// TIA Portal V20 export
DATA_BLOCK "instGetMotorstarterSignals"   // DB91
// stored: InstanceOfName GetMotorstarterSignals, InstanceOfType FB
"GetMotorstarterSignals"
   // VAR_INPUT
   //    Et200SpMotorstarterInterfaceAllUnits { ExternalAccessible := 'False'; ExternalVisible := 'False'; ExternalWritable := 'False'} : Array[0.."NO_OF_UNITS"] of "typeEmMotorStarterInterface";
   //    numberOfMS : USInt := 1;
   // END_VAR
   // VAR_OUTPUT
   //    selectedUnit : USInt := 1;
   //    selectedEM : USInt := 6;
   //    error : Word := 16#7001;
   // END_VAR
   // VAR_IN_OUT
   //    Et200SpMotorstarterInterfaceHmi : "typeEt200SpMotorstarterInterfaceHmi";
   // END_VAR
   // VAR
   //    statSelectedEMMotorStarter : USInt := 6;
   //    statSelectedUnitMotorStarter : USInt := 1;
   // END_VAR
BEGIN
   Et200SpMotorstarterInterfaceAllUnits[0].EMmotorstarter[0].et200SpMotorstarterCurrent[0..1] := 0.0;
   Et200SpMotorstarterInterfaceAllUnits[0].EMmotorstarter[1].et200SpMotorstarterCurrent[0..1] := 0.0;
   Et200SpMotorstarterInterfaceAllUnits[0].EMmotorstarter[2].et200SpMotorstarterCurrent[0..1] := 0.0;
   Et200SpMotorstarterInterfaceAllUnits[0].EMmotorstarter[3].et200SpMotorstarterCurrent[0..1] := 0.0;
   Et200SpMotorstarterInterfaceAllUnits[0].EMmotorstarter[4].et200SpMotorstarterCurrent[0..1] := 0.0;
   Et200SpMotorstarterInterfaceAllUnits[0].EMmotorstarter[5].et200SpMotorstarterCurrent[0..1] := 0.0;
   Et200SpMotorstarterInterfaceAllUnits[0].EMmotorstarter[6].et200SpMotorstarterCurrent[0..1] := 0.0;
   Et200SpMotorstarterInterfaceAllUnits[0].EMmotorstarter[7].et200SpMotorstarterCurrent[0..1] := 0.0;
   Et200SpMotorstarterInterfaceAllUnits[0].EMmotorstarter[0].et200SpMotorstarterInputs[0..1].readyAutomatic := FALSE;
   Et200SpMotorstarterInterfaceAllUnits[0].EMmotorstarter[1].et200SpMotorstarterInputs[0..1].readyAutomatic := FALSE;
   Et200SpMotorstarterInterfaceAllUnits[0].EMmotorstarter[2].et200SpMotorstarterInputs[0..1].readyAutomatic := FALSE;
   Et200SpMotorstarterInterfaceAllUnits[0].EMmotorstarter[3].et200SpMotorstarterInputs[0..1].readyAutomatic := FALSE;
   Et200SpMotorstarterInterfaceAllUnits[0].EMmotorstarter[4].et200SpMotorstarterInputs[0..1].readyAutomatic := FALSE;
   Et200SpMotorstarterInterfaceAllUnits[0].EMmotorstarter[5].et200SpMotorstarterInputs[0..1].readyAutomatic := FALSE;
   Et200SpMotorstarterInterfaceAllUnits[0].EMmotorstarter[6].et200SpMotorstarterInputs[0..1].readyAutomatic := FALSE;
   Et200SpMotorstarterInterfaceAllUnits[0].EMmotorstarter[7].et200SpMotorstarterInputs[0..1].readyAutomatic := FALSE;
   Et200SpMotorstarterInterfaceAllUnits[0].EMmotorstarter[0].et200SpMotorstarterInputs[0..1].motorOn := FALSE;
   Et200SpMotorstarterInterfaceAllUnits[0].EMmotorstarter[1].et200SpMotorstarterInputs[0..1].motorOn := FALSE;
   Et200SpMotorstarterInterfaceAllUnits[0].EMmotorstarter[2].et200SpMotorstarterInputs[0..1].motorOn := FALSE;
   Et200SpMotorstarterInterfaceAllUnits[0].EMmotorstarter[3].et200SpMotorstarterInputs[0..1].motorOn := FALSE;
   Et200SpMotorstarterInterfaceAllUnits[0].EMmotorstarter[4].et200SpMotorstarterInputs[0..1].motorOn := FALSE;
   Et200SpMotorstarterInterfaceAllUnits[0].EMmotorstarter[5].et200SpMotorstarterInputs[0..1].motorOn := FALSE;
   Et200SpMotorstarterInterfaceAllUnits[0].EMmotorstarter[6].et200SpMotorstarterInputs[0..1].motorOn := FALSE;
   Et200SpMotorstarterInterfaceAllUnits[0].EMmotorstarter[7].et200SpMotorstarterInputs[0..1].motorOn := FALSE;
   Et200SpMotorstarterInterfaceAllUnits[0].EMmotorstarter[0].et200SpMotorstarterInputs[0..1].groupFault := FALSE;
   Et200SpMotorstarterInterfaceAllUnits[0].EMmotorstarter[1].et200SpMotorstarterInputs[0..1].groupFault := FALSE;
   Et200SpMotorstarterInterfaceAllUnits[0].EMmotorstarter[2].et200SpMotorstarterInputs[0..1].groupFault := FALSE;
   Et200SpMotorstarterInterfaceAllUnits[0].EMmotorstarter[3].et200SpMotorstarterInputs[0..1].groupFault := FALSE;
   Et200SpMotorstarterInterfaceAllUnits[0].EMmotorstarter[4].et200SpMotorstarterInputs[0..1].groupFault := FALSE;
   Et200SpMotorstarterInterfaceAllUnits[0].EMmotorstarter[5].et200SpMotorstarterInputs[0..1].groupFault := FALSE;
   Et200SpMotorstarterInterfaceAllUnits[0].EMmotorstarter[6].et200SpMotorstarterInputs[0..1].groupFault := FALSE;
   Et200SpMotorstarterInterfaceAllUnits[0].EMmotorstarter[7].et200SpMotorstarterInputs[0..1].groupFault := FALSE;
   Et200SpMotorstarterInterfaceAllUnits[0].EMmotorstarter[0].et200SpMotorstarterInputs[0..1].groupWarning := FALSE;
   Et200SpMotorstarterInterfaceAllUnits[0].EMmotorstarter[1].et200SpMotorstarterInputs[0..1].groupWarning := FALSE;
   Et200SpMotorstarterInterfaceAllUnits[0].EMmotorstarter[2].et200SpMotorstarterInputs[0..1].groupWarning := FALSE;
   Et200SpMotorstarterInterfaceAllUnits[0].EMmotorstarter[3].et200SpMotorstarterInputs[0..1].groupWarning := FALSE;
   Et200SpMotorstarterInterfaceAllUnits[0].EMmotorstarter[4].et200SpMotorstarterInputs[0..1].groupWarning := FALSE;
   Et200SpMotorstarterInterfaceAllUnits[0].EMmotorstarter[5].et200SpMotorstarterInputs[0..1].groupWarning := FALSE;
   Et200SpMotorstarterInterfaceAllUnits[0].EMmotorstarter[6].et200SpMotorstarterInputs[0..1].groupWarning := FALSE;
   Et200SpMotorstarterInterfaceAllUnits[0].EMmotorstarter[7].et200SpMotorstarterInputs[0..1].groupWarning := FALSE;
   Et200SpMotorstarterInterfaceAllUnits[0].EMmotorstarter[0].et200SpMotorstarterInputs[0..1].input1 := FALSE;
   Et200SpMotorstarterInterfaceAllUnits[0].EMmotorstarter[1].et200SpMotorstarterInputs[0..1].input1 := FALSE;
   Et200SpMotorstarterInterfaceAllUnits[0].EMmotorstarter[2].et200SpMotorstarterInputs[0..1].input1 := FALSE;
   Et200SpMotorstarterInterfaceAllUnits[0].EMmotorstarter[3].et200SpMotorstarterInputs[0..1].input1 := FALSE;
   Et200SpMotorstarterInterfaceAllUnits[0].EMmotorstarter[4].et200SpMotorstarterInputs[0..1].input1 := FALSE;
   Et200SpMotorstarterInterfaceAllUnits[0].EMmotorstarter[5].et200SpMotorstarterInputs[0..1].input1 := FALSE;
   Et200SpMotorstarterInterfaceAllUnits[0].EMmotorstarter[6].et200SpMotorstarterInputs[0..1].input1 := FALSE;
   Et200SpMotorstarterInterfaceAllUnits[0].EMmotorstarter[7].et200SpMotorstarterInputs[0..1].input1 := FALSE;
   Et200SpMotorstarterInterfaceAllUnits[0].EMmotorstarter[0].et200SpMotorstarterInputs[0..1].input2 := FALSE;
   Et200SpMotorstarterInterfaceAllUnits[0].EMmotorstarter[1].et200SpMotorstarterInputs[0..1].input2 := FALSE;
   Et200SpMotorstarterInterfaceAllUnits[0].EMmotorstarter[2].et200SpMotorstarterInputs[0..1].input2 := FALSE;
   Et200SpMotorstarterInterfaceAllUnits[0].EMmotorstarter[3].et200SpMotorstarterInputs[0..1].input2 := FALSE;
   Et200SpMotorstarterInterfaceAllUnits[0].EMmotorstarter[4].et200SpMotorstarterInputs[0..1].input2 := FALSE;
   Et200SpMotorstarterInterfaceAllUnits[0].EMmotorstarter[5].et200SpMotorstarterInputs[0..1].input2 := FALSE;
   Et200SpMotorstarterInterfaceAllUnits[0].EMmotorstarter[6].et200SpMotorstarterInputs[0..1].input2 := FALSE;
   Et200SpMotorstarterInterfaceAllUnits[0].EMmotorstarter[7].et200SpMotorstarterInputs[0..1].input2 := FALSE;
   Et200SpMotorstarterInterfaceAllUnits[0].EMmotorstarter[0].et200SpMotorstarterInputs[0..1].input3 := FALSE;
   Et200SpMotorstarterInterfaceAllUnits[0].EMmotorstarter[1].et200SpMotorstarterInputs[0..1].input3 := FALSE;
   Et200SpMotorstarterInterfaceAllUnits[0].EMmotorstarter[2].et200SpMotorstarterInputs[0..1].input3 := FALSE;
   Et200SpMotorstarterInterfaceAllUnits[0].EMmotorstarter[3].et200SpMotorstarterInputs[0..1].input3 := FALSE;
   Et200SpMotorstarterInterfaceAllUnits[0].EMmotorstarter[4].et200SpMotorstarterInputs[0..1].input3 := FALSE;
   Et200SpMotorstarterInterfaceAllUnits[0].EMmotorstarter[5].et200SpMotorstarterInputs[0..1].input3 := FALSE;
   Et200SpMotorstarterInterfaceAllUnits[0].EMmotorstarter[6].et200SpMotorstarterInputs[0..1].input3 := FALSE;
   Et200SpMotorstarterInterfaceAllUnits[0].EMmotorstarter[7].et200SpMotorstarterInputs[0..1].input3 := FALSE;
   Et200SpMotorstarterInterfaceAllUnits[0].EMmotorstarter[0].et200SpMotorstarterInputs[0..1].inputLocalCtrl := FALSE;
   Et200SpMotorstarterInterfaceAllUnits[0].EMmotorstarter[1].et200SpMotorstarterInputs[0..1].inputLocalCtrl := FALSE;
   Et200SpMotorstarterInterfaceAllUnits[0].EMmotorstarter[2].et200SpMotorstarterInputs[0..1].inputLocalCtrl := FALSE;
   Et200SpMotorstarterInterfaceAllUnits[0].EMmotorstarter[3].et200SpMotorstarterInputs[0..1].inputLocalCtrl := FALSE;
   Et200SpMotorstarterInterfaceAllUnits[0].EMmotorstarter[4].et200SpMotorstarterInputs[0..1].inputLocalCtrl := FALSE;
   Et200SpMotorstarterInterfaceAllUnits[0].EMmotorstarter[5].et200SpMotorstarterInputs[0..1].inputLocalCtrl := FALSE;
   Et200SpMotorstarterInterfaceAllUnits[0].EMmotorstarter[6].et200SpMotorstarterInputs[0..1].inputLocalCtrl := FALSE;
   Et200SpMotorstarterInterfaceAllUnits[0].EMmotorstarter[7].et200SpMotorstarterInputs[0..1].inputLocalCtrl := FALSE;
   Et200SpMotorstarterInterfaceAllUnits[0].EMmotorstarter[0].et200SpMotorstarterInputs[0..1].iActBit0 := FALSE;
   Et200SpMotorstarterInterfaceAllUnits[0].EMmotorstarter[1].et200SpMotorstarterInputs[0..1].iActBit0 := FALSE;
   Et200SpMotorstarterInterfaceAllUnits[0].EMmotorstarter[2].et200SpMotorstarterInputs[0..1].iActBit0 := FALSE;
   Et200SpMotorstarterInterfaceAllUnits[0].EMmotorstarter[3].et200SpMotorstarterInputs[0..1].iActBit0 := FALSE;
   Et200SpMotorstarterInterfaceAllUnits[0].EMmotorstarter[4].et200SpMotorstarterInputs[0..1].iActBit0 := FALSE;
   Et200SpMotorstarterInterfaceAllUnits[0].EMmotorstarter[5].et200SpMotorstarterInputs[0..1].iActBit0 := FALSE;
   Et200SpMotorstarterInterfaceAllUnits[0].EMmotorstarter[6].et200SpMotorstarterInputs[0..1].iActBit0 := FALSE;
   Et200SpMotorstarterInterfaceAllUnits[0].EMmotorstarter[7].et200SpMotorstarterInputs[0..1].iActBit0 := FALSE;
   Et200SpMotorstarterInterfaceAllUnits[0].EMmotorstarter[0].et200SpMotorstarterInputs[0..1].iActBit1 := FALSE;
   Et200SpMotorstarterInterfaceAllUnits[0].EMmotorstarter[1].et200SpMotorstarterInputs[0..1].iActBit1 := FALSE;
   Et200SpMotorstarterInterfaceAllUnits[0].EMmotorstarter[2].et200SpMotorstarterInputs[0..1].iActBit1 := FALSE;
   Et200SpMotorstarterInterfaceAllUnits[0].EMmotorstarter[3].et200SpMotorstarterInputs[0..1].iActBit1 := FALSE;
   Et200SpMotorstarterInterfaceAllUnits[0].EMmotorstarter[4].et200SpMotorstarterInputs[0..1].iActBit1 := FALSE;
   Et200SpMotorstarterInterfaceAllUnits[0].EMmotorstarter[5].et200SpMotorstarterInputs[0..1].iActBit1 := FALSE;
   Et200SpMotorstarterInterfaceAllUnits[0].EMmotorstarter[6].et200SpMotorstarterInputs[0..1].iActBit1 := FALSE;
   Et200SpMotorstarterInterfaceAllUnits[0].EMmotorstarter[7].et200SpMotorstarterInputs[0..1].iActBit1 := FALSE;
   Et200SpMotorstarterInterfaceAllUnits[0].EMmotorstarter[0].et200SpMotorstarterInputs[0..1].iActBit2 := FALSE;
   Et200SpMotorstarterInterfaceAllUnits[0].EMmotorstarter[1].et200SpMotorstarterInputs[0..1].iActBit2 := FALSE;
   Et200SpMotorstarterInterfaceAllUnits[0].EMmotorstarter[2].et200SpMotorstarterInputs[0..1].iActBit2 := FALSE;
   Et200SpMotorstarterInterfaceAllUnits[0].EMmotorstarter[3].et200SpMotorstarterInputs[0..1].iActBit2 := FALSE;
   Et200SpMotorstarterInterfaceAllUnits[0].EMmotorstarter[4].et200SpMotorstarterInputs[0..1].iActBit2 := FALSE;
   Et200SpMotorstarterInterfaceAllUnits[0].EMmotorstarter[5].et200SpMotorstarterInputs[0..1].iActBit2 := FALSE;
   Et200SpMotorstarterInterfaceAllUnits[0].EMmotorstarter[6].et200SpMotorstarterInputs[0..1].iActBit2 := FALSE;
   Et200SpMotorstarterInterfaceAllUnits[0].EMmotorstarter[7].et200SpMotorstarterInputs[0..1].iActBit2 := FALSE;
   Et200SpMotorstarterInterfaceAllUnits[0].EMmotorstarter[0].et200SpMotorstarterInputs[0..1].iActBit3 := FALSE;
   Et200SpMotorstarterInterfaceAllUnits[0].EMmotorstarter[1].et200SpMotorstarterInputs[0..1].iActBit3 := FALSE;
   Et200SpMotorstarterInterfaceAllUnits[0].EMmotorstarter[2].et200SpMotorstarterInputs[0..1].iActBit3 := FALSE;
   Et200SpMotorstarterInterfaceAllUnits[0].EMmotorstarter[3].et200SpMotorstarterInputs[0..1].iActBit3 := FALSE;
   Et200SpMotorstarterInterfaceAllUnits[0].EMmotorstarter[4].et200SpMotorstarterInputs[0..1].iActBit3 := FALSE;
   Et200SpMotorstarterInterfaceAllUnits[0].EMmotorstarter[5].et200SpMotorstarterInputs[0..1].iActBit3 := FALSE;
   Et200SpMotorstarterInterfaceAllUnits[0].EMmotorstarter[6].et200SpMotorstarterInputs[0..1].iActBit3 := FALSE;
   Et200SpMotorstarterInterfaceAllUnits[0].EMmotorstarter[7].et200SpMotorstarterInputs[0..1].iActBit3 := FALSE;
   Et200SpMotorstarterInterfaceAllUnits[0].EMmotorstarter[0].et200SpMotorstarterInputs[0..1].iActBit4 := FALSE;
   Et200SpMotorstarterInterfaceAllUnits[0].EMmotorstarter[1].et200SpMotorstarterInputs[0..1].iActBit4 := FALSE;
   Et200SpMotorstarterInterfaceAllUnits[0].EMmotorstarter[2].et200SpMotorstarterInputs[0..1].iActBit4 := FALSE;
   Et200SpMotorstarterInterfaceAllUnits[0].EMmotorstarter[3].et200SpMotorstarterInputs[0..1].iActBit4 := FALSE;
   Et200SpMotorstarterInterfaceAllUnits[0].EMmotorstarter[4].et200SpMotorstarterInputs[0..1].iActBit4 := FALSE;
   Et200SpMotorstarterInterfaceAllUnits[0].EMmotorstarter[5].et200SpMotorstarterInputs[0..1].iActBit4 := FALSE;
   Et200SpMotorstarterInterfaceAllUnits[0].EMmotorstarter[6].et200SpMotorstarterInputs[0..1].iActBit4 := FALSE;
   Et200SpMotorstarterInterfaceAllUnits[0].EMmotorstarter[7].et200SpMotorstarterInputs[0..1].iActBit4 := FALSE;
   Et200SpMotorstarterInterfaceAllUnits[0].EMmotorstarter[0].et200SpMotorstarterInputs[0..1].iActBit5 := FALSE;
   Et200SpMotorstarterInterfaceAllUnits[0].EMmotorstarter[1].et200SpMotorstarterInputs[0..1].iActBit5 := FALSE;
   Et200SpMotorstarterInterfaceAllUnits[0].EMmotorstarter[2].et200SpMotorstarterInputs[0..1].iActBit5 := FALSE;
   Et200SpMotorstarterInterfaceAllUnits[0].EMmotorstarter[3].et200SpMotorstarterInputs[0..1].iActBit5 := FALSE;
   Et200SpMotorstarterInterfaceAllUnits[0].EMmotorstarter[4].et200SpMotorstarterInputs[0..1].iActBit5 := FALSE;
   Et200SpMotorstarterInterfaceAllUnits[0].EMmotorstarter[5].et200SpMotorstarterInputs[0..1].iActBit5 := FALSE;
   Et200SpMotorstarterInterfaceAllUnits[0].EMmotorstarter[6].et200SpMotorstarterInputs[0..1].iActBit5 := FALSE;
   Et200SpMotorstarterInterfaceAllUnits[0].EMmotorstarter[7].et200SpMotorstarterInputs[0..1].iActBit5 := FALSE;
   Et200SpMotorstarterInterfaceAllUnits[0].EMmotorstarter[0].et200SpMotorstarterInputs[0..1].manualOperating := FALSE;
   Et200SpMotorstarterInterfaceAllUnits[0].EMmotorstarter[1].et200SpMotorstarterInputs[0..1].manualOperating := FALSE;
   Et200SpMotorstarterInterfaceAllUnits[0].EMmotorstarter[2].et200SpMotorstarterInputs[0..1].manualOperating := FALSE;
   Et200SpMotorstarterInterfaceAllUnits[0].EMmotorstarter[3].et200SpMotorstarterInputs[0..1].manualOperating := FALSE;
   Et200SpMotorstarterInterfaceAllUnits[0].EMmotorstarter[4].et200SpMotorstarterInputs[0..1].manualOperating := FALSE;
   Et200SpMotorstarterInterfaceAllUnits[0].EMmotorstarter[5].et200SpMotorstarterInputs[0..1].manualOperating := FALSE;
   Et200SpMotorstarterInterfaceAllUnits[0].EMmotorstarter[6].et200SpMotorstarterInputs[0..1].manualOperating := FALSE;
   Et200SpMotorstarterInterfaceAllUnits[0].EMmotorstarter[7].et200SpMotorstarterInputs[0..1].manualOperating := FALSE;
   Et200SpMotorstarterInterfaceAllUnits[0].EMmotorstarter[0].et200SpMotorstarterInputs[0..1].spare1 := FALSE;
   Et200SpMotorstarterInterfaceAllUnits[0].EMmotorstarter[1].et200SpMotorstarterInputs[0..1].spare1 := FALSE;
   Et200SpMotorstarterInterfaceAllUnits[0].EMmotorstarter[2].et200SpMotorstarterInputs[0..1].spare1 := FALSE;
   Et200SpMotorstarterInterfaceAllUnits[0].EMmotorstarter[3].et200SpMotorstarterInputs[0..1].spare1 := FALSE;
   Et200SpMotorstarterInterfaceAllUnits[0].EMmotorstarter[4].et200SpMotorstarterInputs[0..1].spare1 := FALSE;
   Et200SpMotorstarterInterfaceAllUnits[0].EMmotorstarter[5].et200SpMotorstarterInputs[0..1].spare1 := FALSE;
   Et200SpMotorstarterInterfaceAllUnits[0].EMmotorstarter[6].et200SpMotorstarterInputs[0..1].spare1 := FALSE;
   Et200SpMotorstarterInterfaceAllUnits[0].EMmotorstarter[7].et200SpMotorstarterInputs[0..1].spare1 := FALSE;
   Et200SpMotorstarterInterfaceAllUnits[0].EMmotorstarter[0].et200SpMotorstarterInputs[0..1].readyStartOn := FALSE;
   Et200SpMotorstarterInterfaceAllUnits[0].EMmotorstarter[1].et200SpMotorstarterInputs[0..1].readyStartOn := FALSE;
   Et200SpMotorstarterInterfaceAllUnits[0].EMmotorstarter[2].et200SpMotorstarterInputs[0..1].readyStartOn := FALSE;
   Et200SpMotorstarterInterfaceAllUnits[0].EMmotorstarter[3].et200SpMotorstarterInputs[0..1].readyStartOn := FALSE;
   Et200SpMotorstarterInterfaceAllUnits[0].EMmotorstarter[4].et200SpMotorstarterInputs[0..1].readyStartOn := FALSE;
   Et200SpMotorstarterInterfaceAllUnits[0].EMmotorstarter[5].et200SpMotorstarterInputs[0..1].readyStartOn := FALSE;
   Et200SpMotorstarterInterfaceAllUnits[0].EMmotorstarter[6].et200SpMotorstarterInputs[0..1].readyStartOn := FALSE;
   Et200SpMotorstarterInterfaceAllUnits[0].EMmotorstarter[7].et200SpMotorstarterInputs[0..1].readyStartOn := FALSE;
   Et200SpMotorstarterInterfaceAllUnits[0].EMmotorstarter[0].et200SpMotorstarterInputs[0..1].motorOnRight := FALSE;
   Et200SpMotorstarterInterfaceAllUnits[0].EMmotorstarter[1].et200SpMotorstarterInputs[0..1].motorOnRight := FALSE;
   Et200SpMotorstarterInterfaceAllUnits[0].EMmotorstarter[2].et200SpMotorstarterInputs[0..1].motorOnRight := FALSE;
   Et200SpMotorstarterInterfaceAllUnits[0].EMmotorstarter[3].et200SpMotorstarterInputs[0..1].motorOnRight := FALSE;
   Et200SpMotorstarterInterfaceAllUnits[0].EMmotorstarter[4].et200SpMotorstarterInputs[0..1].motorOnRight := FALSE;
   Et200SpMotorstarterInterfaceAllUnits[0].EMmotorstarter[5].et200SpMotorstarterInputs[0..1].motorOnRight := FALSE;
   Et200SpMotorstarterInterfaceAllUnits[0].EMmotorstarter[6].et200SpMotorstarterInputs[0..1].motorOnRight := FALSE;
   Et200SpMotorstarterInterfaceAllUnits[0].EMmotorstarter[7].et200SpMotorstarterInputs[0..1].motorOnRight := FALSE;
   Et200SpMotorstarterInterfaceAllUnits[0].EMmotorstarter[0].et200SpMotorstarterInputs[0..1].motorOnLeft := FALSE;
   Et200SpMotorstarterInterfaceAllUnits[0].EMmotorstarter[1].et200SpMotorstarterInputs[0..1].motorOnLeft := FALSE;
   Et200SpMotorstarterInterfaceAllUnits[0].EMmotorstarter[2].et200SpMotorstarterInputs[0..1].motorOnLeft := FALSE;
   Et200SpMotorstarterInterfaceAllUnits[0].EMmotorstarter[3].et200SpMotorstarterInputs[0..1].motorOnLeft := FALSE;
   Et200SpMotorstarterInterfaceAllUnits[0].EMmotorstarter[4].et200SpMotorstarterInputs[0..1].motorOnLeft := FALSE;
   Et200SpMotorstarterInterfaceAllUnits[0].EMmotorstarter[5].et200SpMotorstarterInputs[0..1].motorOnLeft := FALSE;
   Et200SpMotorstarterInterfaceAllUnits[0].EMmotorstarter[6].et200SpMotorstarterInputs[0..1].motorOnLeft := FALSE;
   Et200SpMotorstarterInterfaceAllUnits[0].EMmotorstarter[7].et200SpMotorstarterInputs[0..1].motorOnLeft := FALSE;
   Et200SpMotorstarterInterfaceAllUnits[0].EMmotorstarter[0].et200SpMotorstarterInputs[0..1].quickstopActive := FALSE;
   Et200SpMotorstarterInterfaceAllUnits[0].EMmotorstarter[1].et200SpMotorstarterInputs[0..1].quickstopActive := FALSE;
   Et200SpMotorstarterInterfaceAllUnits[0].EMmotorstarter[2].et200SpMotorstarterInputs[0..1].quickstopActive := FALSE;
   Et200SpMotorstarterInterfaceAllUnits[0].EMmotorstarter[3].et200SpMotorstarterInputs[0..1].quickstopActive := FALSE;
   Et200SpMotorstarterInterfaceAllUnits[0].EMmotorstarter[4].et200SpMotorstarterInputs[0..1].quickstopActive := FALSE;
   Et200SpMotorstarterInterfaceAllUnits[0].EMmotorstarter[5].et200SpMotorstarterInputs[0..1].quickstopActive := FALSE;
   Et200SpMotorstarterInterfaceAllUnits[0].EMmotorstarter[6].et200SpMotorstarterInputs[0..1].quickstopActive := FALSE;
   Et200SpMotorstarterInterfaceAllUnits[0].EMmotorstarter[7].et200SpMotorstarterInputs[0..1].quickstopActive := FALSE;
   Et200SpMotorstarterInterfaceAllUnits[0].EMmotorstarter[0].et200SpMotorstarterInputs[0..1].energySaving := FALSE;
   Et200SpMotorstarterInterfaceAllUnits[0].EMmotorstarter[1].et200SpMotorstarterInputs[0..1].energySaving := FALSE;
   Et200SpMotorstarterInterfaceAllUnits[0].EMmotorstarter[2].et200SpMotorstarterInputs[0..1].energySaving := FALSE;
   Et200SpMotorstarterInterfaceAllUnits[0].EMmotorstarter[3].et200SpMotorstarterInputs[0..1].energySaving := FALSE;
   Et200SpMotorstarterInterfaceAllUnits[0].EMmotorstarter[4].et200SpMotorstarterInputs[0..1].energySaving := FALSE;
   Et200SpMotorstarterInterfaceAllUnits[0].EMmotorstarter[5].et200SpMotorstarterInputs[0..1].energySaving := FALSE;
   Et200SpMotorstarterInterfaceAllUnits[0].EMmotorstarter[6].et200SpMotorstarterInputs[0..1].energySaving := FALSE;
   Et200SpMotorstarterInterfaceAllUnits[0].EMmotorstarter[7].et200SpMotorstarterInputs[0..1].energySaving := FALSE;
   Et200SpMotorstarterInterfaceAllUnits[0].EMmotorstarter[0].et200SpMotorstarterInputs[0..1].moduleInserted := FALSE;
   Et200SpMotorstarterInterfaceAllUnits[0].EMmotorstarter[1].et200SpMotorstarterInputs[0..1].moduleInserted := FALSE;
   Et200SpMotorstarterInterfaceAllUnits[0].EMmotorstarter[2].et200SpMotorstarterInputs[0..1].moduleInserted := FALSE;
   Et200SpMotorstarterInterfaceAllUnits[0].EMmotorstarter[3].et200SpMotorstarterInputs[0..1].moduleInserted := FALSE;
   Et200SpMotorstarterInterfaceAllUnits[0].EMmotorstarter[4].et200SpMotorstarterInputs[0..1].moduleInserted := FALSE;
   Et200SpMotorstarterInterfaceAllUnits[0].EMmotorstarter[5].et200SpMotorstarterInputs[0..1].moduleInserted := FALSE;
   Et200SpMotorstarterInterfaceAllUnits[0].EMmotorstarter[6].et200SpMotorstarterInputs[0..1].moduleInserted := FALSE;
   Et200SpMotorstarterInterfaceAllUnits[0].EMmotorstarter[7].et200SpMotorstarterInputs[0..1].moduleInserted := FALSE;
   Et200SpMotorstarterInterfaceAllUnits[0].EMmotorstarter[0].et200SpMotorstarterInputs[0..1].exProtectionMotorActive := FALSE;
   Et200SpMotorstarterInterfaceAllUnits[0].EMmotorstarter[1].et200SpMotorstarterInputs[0..1].exProtectionMotorActive := FALSE;
   Et200SpMotorstarterInterfaceAllUnits[0].EMmotorstarter[2].et200SpMotorstarterInputs[0..1].exProtectionMotorActive := FALSE;
   Et200SpMotorstarterInterfaceAllUnits[0].EMmotorstarter[3].et200SpMotorstarterInputs[0..1].exProtectionMotorActive := FALSE;
   Et200SpMotorstarterInterfaceAllUnits[0].EMmotorstarter[4].et200SpMotorstarterInputs[0..1].exProtectionMotorActive := FALSE;
   Et200SpMotorstarterInterfaceAllUnits[0].EMmotorstarter[5].et200SpMotorstarterInputs[0..1].exProtectionMotorActive := FALSE;
   Et200SpMotorstarterInterfaceAllUnits[0].EMmotorstarter[6].et200SpMotorstarterInputs[0..1].exProtectionMotorActive := FALSE;
   Et200SpMotorstarterInterfaceAllUnits[0].EMmotorstarter[7].et200SpMotorstarterInputs[0..1].exProtectionMotorActive := FALSE;
   Et200SpMotorstarterInterfaceAllUnits[0].EMmotorstarter[0].et200SpMotorstarterInputs[0..1].blockActive := FALSE;
   Et200SpMotorstarterInterfaceAllUnits[0].EMmotorstarter[1].et200SpMotorstarterInputs[0..1].blockActive := FALSE;
   Et200SpMotorstarterInterfaceAllUnits[0].EMmotorstarter[2].et200SpMotorstarterInputs[0..1].blockActive := FALSE;
   Et200SpMotorstarterInterfaceAllUnits[0].EMmotorstarter[3].et200SpMotorstarterInputs[0..1].blockActive := FALSE;
   Et200SpMotorstarterInterfaceAllUnits[0].EMmotorstarter[4].et200SpMotorstarterInputs[0..1].blockActive := FALSE;
   Et200SpMotorstarterInterfaceAllUnits[0].EMmotorstarter[5].et200SpMotorstarterInputs[0..1].blockActive := FALSE;
   Et200SpMotorstarterInterfaceAllUnits[0].EMmotorstarter[6].et200SpMotorstarterInputs[0..1].blockActive := FALSE;
   Et200SpMotorstarterInterfaceAllUnits[0].EMmotorstarter[7].et200SpMotorstarterInputs[0..1].blockActive := FALSE;
   Et200SpMotorstarterInterfaceAllUnits[0].EMmotorstarter[0].et200SpMotorstarterInputs[0..1].thermalMotorOverload := FALSE;
   Et200SpMotorstarterInterfaceAllUnits[0].EMmotorstarter[1].et200SpMotorstarterInputs[0..1].thermalMotorOverload := FALSE;
   Et200SpMotorstarterInterfaceAllUnits[0].EMmotorstarter[2].et200SpMotorstarterInputs[0..1].thermalMotorOverload := FALSE;
   Et200SpMotorstarterInterfaceAllUnits[0].EMmotorstarter[3].et200SpMotorstarterInputs[0..1].thermalMotorOverload := FALSE;
   Et200SpMotorstarterInterfaceAllUnits[0].EMmotorstarter[4].et200SpMotorstarterInputs[0..1].thermalMotorOverload := FALSE;
   Et200SpMotorstarterInterfaceAllUnits[0].EMmotorstarter[5].et200SpMotorstarterInputs[0..1].thermalMotorOverload := FALSE;
   Et200SpMotorstarterInterfaceAllUnits[0].EMmotorstarter[6].et200SpMotorstarterInputs[0..1].thermalMotorOverload := FALSE;
   Et200SpMotorstarterInterfaceAllUnits[0].EMmotorstarter[7].et200SpMotorstarterInputs[0..1].thermalMotorOverload := FALSE;
   Et200SpMotorstarterInterfaceAllUnits[0].EMmotorstarter[0].et200SpMotorstarterInputs[0..1].spare5 := FALSE;
   Et200SpMotorstarterInterfaceAllUnits[0].EMmotorstarter[1].et200SpMotorstarterInputs[0..1].spare5 := FALSE;
   Et200SpMotorstarterInterfaceAllUnits[0].EMmotorstarter[2].et200SpMotorstarterInputs[0..1].spare5 := FALSE;
   Et200SpMotorstarterInterfaceAllUnits[0].EMmotorstarter[3].et200SpMotorstarterInputs[0..1].spare5 := FALSE;
   Et200SpMotorstarterInterfaceAllUnits[0].EMmotorstarter[4].et200SpMotorstarterInputs[0..1].spare5 := FALSE;
   Et200SpMotorstarterInterfaceAllUnits[0].EMmotorstarter[5].et200SpMotorstarterInputs[0..1].spare5 := FALSE;
   Et200SpMotorstarterInterfaceAllUnits[0].EMmotorstarter[6].et200SpMotorstarterInputs[0..1].spare5 := FALSE;
   Et200SpMotorstarterInterfaceAllUnits[0].EMmotorstarter[7].et200SpMotorstarterInputs[0..1].spare5 := FALSE;
   Et200SpMotorstarterInterfaceAllUnits[0].EMmotorstarter[0].et200SpMotorstarterInputs[0..1].currentLimitTripping := FALSE;
   Et200SpMotorstarterInterfaceAllUnits[0].EMmotorstarter[1].et200SpMotorstarterInputs[0..1].currentLimitTripping := FALSE;
   Et200SpMotorstarterInterfaceAllUnits[0].EMmotorstarter[2].et200SpMotorstarterInputs[0..1].currentLimitTripping := FALSE;
   Et200SpMotorstarterInterfaceAllUnits[0].EMmotorstarter[3].et200SpMotorstarterInputs[0..1].currentLimitTripping := FALSE;
   Et200SpMotorstarterInterfaceAllUnits[0].EMmotorstarter[4].et200SpMotorstarterInputs[0..1].currentLimitTripping := FALSE;
   Et200SpMotorstarterInterfaceAllUnits[0].EMmotorstarter[5].et200SpMotorstarterInputs[0..1].currentLimitTripping := FALSE;
   Et200SpMotorstarterInterfaceAllUnits[0].EMmotorstarter[6].et200SpMotorstarterInputs[0..1].currentLimitTripping := FALSE;
   Et200SpMotorstarterInterfaceAllUnits[0].EMmotorstarter[7].et200SpMotorstarterInputs[0..1].currentLimitTripping := FALSE;
   Et200SpMotorstarterInterfaceAllUnits[0].EMmotorstarter[0].et200SpMotorstarterInputs[0..1].statusFailDi := FALSE;
   Et200SpMotorstarterInterfaceAllUnits[0].EMmotorstarter[1].et200SpMotorstarterInputs[0..1].statusFailDi := FALSE;
   Et200SpMotorstarterInterfaceAllUnits[0].EMmotorstarter[2].et200SpMotorstarterInputs[0..1].statusFailDi := FALSE;
   Et200SpMotorstarterInterfaceAllUnits[0].EMmotorstarter[3].et200SpMotorstarterInputs[0..1].statusFailDi := FALSE;
   Et200SpMotorstarterInterfaceAllUnits[0].EMmotorstarter[4].et200SpMotorstarterInputs[0..1].statusFailDi := FALSE;
   Et200SpMotorstarterInterfaceAllUnits[0].EMmotorstarter[5].et200SpMotorstarterInputs[0..1].statusFailDi := FALSE;
   Et200SpMotorstarterInterfaceAllUnits[0].EMmotorstarter[6].et200SpMotorstarterInputs[0..1].statusFailDi := FALSE;
   Et200SpMotorstarterInterfaceAllUnits[0].EMmotorstarter[7].et200SpMotorstarterInputs[0..1].statusFailDi := FALSE;
   Et200SpMotorstarterInterfaceAllUnits[0].EMmotorstarter[0].et200SpMotorstarterInputs[0..1].residualCurrent := FALSE;
   Et200SpMotorstarterInterfaceAllUnits[0].EMmotorstarter[1].et200SpMotorstarterInputs[0..1].residualCurrent := FALSE;
   Et200SpMotorstarterInterfaceAllUnits[0].EMmotorstarter[2].et200SpMotorstarterInputs[0..1].residualCurrent := FALSE;
   Et200SpMotorstarterInterfaceAllUnits[0].EMmotorstarter[3].et200SpMotorstarterInputs[0..1].residualCurrent := FALSE;
   Et200SpMotorstarterInterfaceAllUnits[0].EMmotorstarter[4].et200SpMotorstarterInputs[0..1].residualCurrent := FALSE;
   Et200SpMotorstarterInterfaceAllUnits[0].EMmotorstarter[5].et200SpMotorstarterInputs[0..1].residualCurrent := FALSE;
   Et200SpMotorstarterInterfaceAllUnits[0].EMmotorstarter[6].et200SpMotorstarterInputs[0..1].residualCurrent := FALSE;
   Et200SpMotorstarterInterfaceAllUnits[0].EMmotorstarter[7].et200SpMotorstarterInputs[0..1].residualCurrent := FALSE;
   Et200SpMotorstarterInterfaceAllUnits[0].EMmotorstarter[0].et200SpMotorstarterInputs[0..1].asymmetryDetected := FALSE;
   Et200SpMotorstarterInterfaceAllUnits[0].EMmotorstarter[1].et200SpMotorstarterInputs[0..1].asymmetryDetected := FALSE;
   Et200SpMotorstarterInterfaceAllUnits[0].EMmotorstarter[2].et200SpMotorstarterInputs[0..1].asymmetryDetected := FALSE;
   Et200SpMotorstarterInterfaceAllUnits[0].EMmotorstarter[3].et200SpMotorstarterInputs[0..1].asymmetryDetected := FALSE;
   Et200SpMotorstarterInterfaceAllUnits[0].EMmotorstarter[4].et200SpMotorstarterInputs[0..1].asymmetryDetected := FALSE;
   Et200SpMotorstarterInterfaceAllUnits[0].EMmotorstarter[5].et200SpMotorstarterInputs[0..1].asymmetryDetected := FALSE;
   Et200SpMotorstarterInterfaceAllUnits[0].EMmotorstarter[6].et200SpMotorstarterInputs[0..1].asymmetryDetected := FALSE;
   Et200SpMotorstarterInterfaceAllUnits[0].EMmotorstarter[7].et200SpMotorstarterInputs[0..1].asymmetryDetected := FALSE;
   Et200SpMotorstarterInterfaceAllUnits[0].EMmotorstarter[0].et200SpMotorstarterInputs[0..1].overtemperature := FALSE;
   Et200SpMotorstarterInterfaceAllUnits[0].EMmotorstarter[1].et200SpMotorstarterInputs[0..1].overtemperature := FALSE;
   Et200SpMotorstarterInterfaceAllUnits[0].EMmotorstarter[2].et200SpMotorstarterInputs[0..1].overtemperature := FALSE;
   Et200SpMotorstarterInterfaceAllUnits[0].EMmotorstarter[3].et200SpMotorstarterInputs[0..1].overtemperature := FALSE;
   Et200SpMotorstarterInterfaceAllUnits[0].EMmotorstarter[4].et200SpMotorstarterInputs[0..1].overtemperature := FALSE;
   Et200SpMotorstarterInterfaceAllUnits[0].EMmotorstarter[5].et200SpMotorstarterInputs[0..1].overtemperature := FALSE;
   Et200SpMotorstarterInterfaceAllUnits[0].EMmotorstarter[6].et200SpMotorstarterInputs[0..1].overtemperature := FALSE;
   Et200SpMotorstarterInterfaceAllUnits[0].EMmotorstarter[7].et200SpMotorstarterInputs[0..1].overtemperature := FALSE;
   Et200SpMotorstarterInterfaceAllUnits[0].EMmotorstarter[0].et200SpMotorstarterInputs[0..1].spare7 := FALSE;
   Et200SpMotorstarterInterfaceAllUnits[0].EMmotorstarter[1].et200SpMotorstarterInputs[0..1].spare7 := FALSE;
   Et200SpMotorstarterInterfaceAllUnits[0].EMmotorstarter[2].et200SpMotorstarterInputs[0..1].spare7 := FALSE;
   Et200SpMotorstarterInterfaceAllUnits[0].EMmotorstarter[3].et200SpMotorstarterInputs[0..1].spare7 := FALSE;
   Et200SpMotorstarterInterfaceAllUnits[0].EMmotorstarter[4].et200SpMotorstarterInputs[0..1].spare7 := FALSE;
   Et200SpMotorstarterInterfaceAllUnits[0].EMmotorstarter[5].et200SpMotorstarterInputs[0..1].spare7 := FALSE;
   Et200SpMotorstarterInterfaceAllUnits[0].EMmotorstarter[6].et200SpMotorstarterInputs[0..1].spare7 := FALSE;
   Et200SpMotorstarterInterfaceAllUnits[0].EMmotorstarter[7].et200SpMotorstarterInputs[0..1].spare7 := FALSE;
   Et200SpMotorstarterInterfaceAllUnits[0].EMmotorstarter[0].et200SpMotorstarterOutputs[0..1].motorCw := FALSE;
   Et200SpMotorstarterInterfaceAllUnits[0].EMmotorstarter[1].et200SpMotorstarterOutputs[0..1].motorCw := FALSE;
   Et200SpMotorstarterInterfaceAllUnits[0].EMmotorstarter[2].et200SpMotorstarterOutputs[0..1].motorCw := FALSE;
   Et200SpMotorstarterInterfaceAllUnits[0].EMmotorstarter[3].et200SpMotorstarterOutputs[0..1].motorCw := FALSE;
   Et200SpMotorstarterInterfaceAllUnits[0].EMmotorstarter[4].et200SpMotorstarterOutputs[0..1].motorCw := FALSE;
   Et200SpMotorstarterInterfaceAllUnits[0].EMmotorstarter[5].et200SpMotorstarterOutputs[0..1].motorCw := FALSE;
   Et200SpMotorstarterInterfaceAllUnits[0].EMmotorstarter[6].et200SpMotorstarterOutputs[0..1].motorCw := FALSE;
   Et200SpMotorstarterInterfaceAllUnits[0].EMmotorstarter[7].et200SpMotorstarterOutputs[0..1].motorCw := FALSE;
   Et200SpMotorstarterInterfaceAllUnits[0].EMmotorstarter[0].et200SpMotorstarterOutputs[0..1].motorCww := FALSE;
   Et200SpMotorstarterInterfaceAllUnits[0].EMmotorstarter[1].et200SpMotorstarterOutputs[0..1].motorCww := FALSE;
   Et200SpMotorstarterInterfaceAllUnits[0].EMmotorstarter[2].et200SpMotorstarterOutputs[0..1].motorCww := FALSE;
   Et200SpMotorstarterInterfaceAllUnits[0].EMmotorstarter[3].et200SpMotorstarterOutputs[0..1].motorCww := FALSE;
   Et200SpMotorstarterInterfaceAllUnits[0].EMmotorstarter[4].et200SpMotorstarterOutputs[0..1].motorCww := FALSE;
   Et200SpMotorstarterInterfaceAllUnits[0].EMmotorstarter[5].et200SpMotorstarterOutputs[0..1].motorCww := FALSE;
   Et200SpMotorstarterInterfaceAllUnits[0].EMmotorstarter[6].et200SpMotorstarterOutputs[0..1].motorCww := FALSE;
   Et200SpMotorstarterInterfaceAllUnits[0].EMmotorstarter[7].et200SpMotorstarterOutputs[0..1].motorCww := FALSE;
   Et200SpMotorstarterInterfaceAllUnits[0].EMmotorstarter[0].et200SpMotorstarterOutputs[0..1].reserve1 := FALSE;
   Et200SpMotorstarterInterfaceAllUnits[0].EMmotorstarter[1].et200SpMotorstarterOutputs[0..1].reserve1 := FALSE;
   Et200SpMotorstarterInterfaceAllUnits[0].EMmotorstarter[2].et200SpMotorstarterOutputs[0..1].reserve1 := FALSE;
   Et200SpMotorstarterInterfaceAllUnits[0].EMmotorstarter[3].et200SpMotorstarterOutputs[0..1].reserve1 := FALSE;
   Et200SpMotorstarterInterfaceAllUnits[0].EMmotorstarter[4].et200SpMotorstarterOutputs[0..1].reserve1 := FALSE;
   Et200SpMotorstarterInterfaceAllUnits[0].EMmotorstarter[5].et200SpMotorstarterOutputs[0..1].reserve1 := FALSE;
   Et200SpMotorstarterInterfaceAllUnits[0].EMmotorstarter[6].et200SpMotorstarterOutputs[0..1].reserve1 := FALSE;
   Et200SpMotorstarterInterfaceAllUnits[0].EMmotorstarter[7].et200SpMotorstarterOutputs[0..1].reserve1 := FALSE;
   Et200SpMotorstarterInterfaceAllUnits[0].EMmotorstarter[0].et200SpMotorstarterOutputs[0..1].tripReset := FALSE;
   Et200SpMotorstarterInterfaceAllUnits[0].EMmotorstarter[1].et200SpMotorstarterOutputs[0..1].tripReset := FALSE;
   Et200SpMotorstarterInterfaceAllUnits[0].EMmotorstarter[2].et200SpMotorstarterOutputs[0..1].tripReset := FALSE;
   Et200SpMotorstarterInterfaceAllUnits[0].EMmotorstarter[3].et200SpMotorstarterOutputs[0..1].tripReset := FALSE;
   Et200SpMotorstarterInterfaceAllUnits[0].EMmotorstarter[4].et200SpMotorstarterOutputs[0..1].tripReset := FALSE;
   Et200SpMotorstarterInterfaceAllUnits[0].EMmotorstarter[5].et200SpMotorstarterOutputs[0..1].tripReset := FALSE;
   Et200SpMotorstarterInterfaceAllUnits[0].EMmotorstarter[6].et200SpMotorstarterOutputs[0..1].tripReset := FALSE;
   Et200SpMotorstarterInterfaceAllUnits[0].EMmotorstarter[7].et200SpMotorstarterOutputs[0..1].tripReset := FALSE;
   Et200SpMotorstarterInterfaceAllUnits[0].EMmotorstarter[0].et200SpMotorstarterOutputs[0..1].emergencyStart := FALSE;
   Et200SpMotorstarterInterfaceAllUnits[0].EMmotorstarter[1].et200SpMotorstarterOutputs[0..1].emergencyStart := FALSE;
   Et200SpMotorstarterInterfaceAllUnits[0].EMmotorstarter[2].et200SpMotorstarterOutputs[0..1].emergencyStart := FALSE;
   Et200SpMotorstarterInterfaceAllUnits[0].EMmotorstarter[3].et200SpMotorstarterOutputs[0..1].emergencyStart := FALSE;
   Et200SpMotorstarterInterfaceAllUnits[0].EMmotorstarter[4].et200SpMotorstarterOutputs[0..1].emergencyStart := FALSE;
   Et200SpMotorstarterInterfaceAllUnits[0].EMmotorstarter[5].et200SpMotorstarterOutputs[0..1].emergencyStart := FALSE;
   Et200SpMotorstarterInterfaceAllUnits[0].EMmotorstarter[6].et200SpMotorstarterOutputs[0..1].emergencyStart := FALSE;
   Et200SpMotorstarterInterfaceAllUnits[0].EMmotorstarter[7].et200SpMotorstarterOutputs[0..1].emergencyStart := FALSE;
   Et200SpMotorstarterInterfaceAllUnits[0].EMmotorstarter[0].et200SpMotorstarterOutputs[0..1].reserve2 := FALSE;
   Et200SpMotorstarterInterfaceAllUnits[0].EMmotorstarter[1].et200SpMotorstarterOutputs[0..1].reserve2 := FALSE;
   Et200SpMotorstarterInterfaceAllUnits[0].EMmotorstarter[2].et200SpMotorstarterOutputs[0..1].reserve2 := FALSE;
   Et200SpMotorstarterInterfaceAllUnits[0].EMmotorstarter[3].et200SpMotorstarterOutputs[0..1].reserve2 := FALSE;
   Et200SpMotorstarterInterfaceAllUnits[0].EMmotorstarter[4].et200SpMotorstarterOutputs[0..1].reserve2 := FALSE;
   Et200SpMotorstarterInterfaceAllUnits[0].EMmotorstarter[5].et200SpMotorstarterOutputs[0..1].reserve2 := FALSE;
   Et200SpMotorstarterInterfaceAllUnits[0].EMmotorstarter[6].et200SpMotorstarterOutputs[0..1].reserve2 := FALSE;
   Et200SpMotorstarterInterfaceAllUnits[0].EMmotorstarter[7].et200SpMotorstarterOutputs[0..1].reserve2 := FALSE;
   Et200SpMotorstarterInterfaceAllUnits[0].EMmotorstarter[0].et200SpMotorstarterOutputs[0..1].reserve3 := FALSE;
   Et200SpMotorstarterInterfaceAllUnits[0].EMmotorstarter[1].et200SpMotorstarterOutputs[0..1].reserve3 := FALSE;
   Et200SpMotorstarterInterfaceAllUnits[0].EMmotorstarter[2].et200SpMotorstarterOutputs[0..1].reserve3 := FALSE;
   Et200SpMotorstarterInterfaceAllUnits[0].EMmotorstarter[3].et200SpMotorstarterOutputs[0..1].reserve3 := FALSE;
   Et200SpMotorstarterInterfaceAllUnits[0].EMmotorstarter[4].et200SpMotorstarterOutputs[0..1].reserve3 := FALSE;
   Et200SpMotorstarterInterfaceAllUnits[0].EMmotorstarter[5].et200SpMotorstarterOutputs[0..1].reserve3 := FALSE;
   Et200SpMotorstarterInterfaceAllUnits[0].EMmotorstarter[6].et200SpMotorstarterOutputs[0..1].reserve3 := FALSE;
   Et200SpMotorstarterInterfaceAllUnits[0].EMmotorstarter[7].et200SpMotorstarterOutputs[0..1].reserve3 := FALSE;
   Et200SpMotorstarterInterfaceAllUnits[0].EMmotorstarter[0].et200SpMotorstarterOutputs[0..1].coldStart := FALSE;
   Et200SpMotorstarterInterfaceAllUnits[0].EMmotorstarter[1].et200SpMotorstarterOutputs[0..1].coldStart := FALSE;
   Et200SpMotorstarterInterfaceAllUnits[0].EMmotorstarter[2].et200SpMotorstarterOutputs[0..1].coldStart := FALSE;
   Et200SpMotorstarterInterfaceAllUnits[0].EMmotorstarter[3].et200SpMotorstarterOutputs[0..1].coldStart := FALSE;
   Et200SpMotorstarterInterfaceAllUnits[0].EMmotorstarter[4].et200SpMotorstarterOutputs[0..1].coldStart := FALSE;
   Et200SpMotorstarterInterfaceAllUnits[0].EMmotorstarter[5].et200SpMotorstarterOutputs[0..1].coldStart := FALSE;
   Et200SpMotorstarterInterfaceAllUnits[0].EMmotorstarter[6].et200SpMotorstarterOutputs[0..1].coldStart := FALSE;
   Et200SpMotorstarterInterfaceAllUnits[0].EMmotorstarter[7].et200SpMotorstarterOutputs[0..1].coldStart := FALSE;
   Et200SpMotorstarterInterfaceAllUnits[0].EMmotorstarter[0].et200SpMotorstarterOutputs[0..1].reserve4 := FALSE;
   Et200SpMotorstarterInterfaceAllUnits[0].EMmotorstarter[1].et200SpMotorstarterOutputs[0..1].reserve4 := FALSE;
   Et200SpMotorstarterInterfaceAllUnits[0].EMmotorstarter[2].et200SpMotorstarterOutputs[0..1].reserve4 := FALSE;
   Et200SpMotorstarterInterfaceAllUnits[0].EMmotorstarter[3].et200SpMotorstarterOutputs[0..1].reserve4 := FALSE;
   Et200SpMotorstarterInterfaceAllUnits[0].EMmotorstarter[4].et200SpMotorstarterOutputs[0..1].reserve4 := FALSE;
   Et200SpMotorstarterInterfaceAllUnits[0].EMmotorstarter[5].et200SpMotorstarterOutputs[0..1].reserve4 := FALSE;
   Et200SpMotorstarterInterfaceAllUnits[0].EMmotorstarter[6].et200SpMotorstarterOutputs[0..1].reserve4 := FALSE;
   Et200SpMotorstarterInterfaceAllUnits[0].EMmotorstarter[7].et200SpMotorstarterOutputs[0..1].reserve4 := FALSE;
   Et200SpMotorstarterInterfaceAllUnits[0].EMmotorstarter[0].et200SpMotorstarterOutputs[0..1].reserve5 := FALSE;
   Et200SpMotorstarterInterfaceAllUnits[0].EMmotorstarter[1].et200SpMotorstarterOutputs[0..1].reserve5 := FALSE;
   Et200SpMotorstarterInterfaceAllUnits[0].EMmotorstarter[2].et200SpMotorstarterOutputs[0..1].reserve5 := FALSE;
   Et200SpMotorstarterInterfaceAllUnits[0].EMmotorstarter[3].et200SpMotorstarterOutputs[0..1].reserve5 := FALSE;
   Et200SpMotorstarterInterfaceAllUnits[0].EMmotorstarter[4].et200SpMotorstarterOutputs[0..1].reserve5 := FALSE;
   Et200SpMotorstarterInterfaceAllUnits[0].EMmotorstarter[5].et200SpMotorstarterOutputs[0..1].reserve5 := FALSE;
   Et200SpMotorstarterInterfaceAllUnits[0].EMmotorstarter[6].et200SpMotorstarterOutputs[0..1].reserve5 := FALSE;
   Et200SpMotorstarterInterfaceAllUnits[0].EMmotorstarter[7].et200SpMotorstarterOutputs[0..1].reserve5 := FALSE;
   Et200SpMotorstarterInterfaceAllUnits[0].EMmotorstarter[0].et200SpMotorstarterOutputs[0..1].reserve6 := FALSE;
   Et200SpMotorstarterInterfaceAllUnits[0].EMmotorstarter[1].et200SpMotorstarterOutputs[0..1].reserve6 := FALSE;
   Et200SpMotorstarterInterfaceAllUnits[0].EMmotorstarter[2].et200SpMotorstarterOutputs[0..1].reserve6 := FALSE;
   Et200SpMotorstarterInterfaceAllUnits[0].EMmotorstarter[3].et200SpMotorstarterOutputs[0..1].reserve6 := FALSE;
   Et200SpMotorstarterInterfaceAllUnits[0].EMmotorstarter[4].et200SpMotorstarterOutputs[0..1].reserve6 := FALSE;
   Et200SpMotorstarterInterfaceAllUnits[0].EMmotorstarter[5].et200SpMotorstarterOutputs[0..1].reserve6 := FALSE;
   Et200SpMotorstarterInterfaceAllUnits[0].EMmotorstarter[6].et200SpMotorstarterOutputs[0..1].reserve6 := FALSE;
   Et200SpMotorstarterInterfaceAllUnits[0].EMmotorstarter[7].et200SpMotorstarterOutputs[0..1].reserve6 := FALSE;
   Et200SpMotorstarterInterfaceAllUnits[0].EMmotorstarter[0].et200SpMotorstarterOutputs[0..1].reserve7 := FALSE;
   Et200SpMotorstarterInterfaceAllUnits[0].EMmotorstarter[1].et200SpMotorstarterOutputs[0..1].reserve7 := FALSE;
   Et200SpMotorstarterInterfaceAllUnits[0].EMmotorstarter[2].et200SpMotorstarterOutputs[0..1].reserve7 := FALSE;
   Et200SpMotorstarterInterfaceAllUnits[0].EMmotorstarter[3].et200SpMotorstarterOutputs[0..1].reserve7 := FALSE;
   Et200SpMotorstarterInterfaceAllUnits[0].EMmotorstarter[4].et200SpMotorstarterOutputs[0..1].reserve7 := FALSE;
   Et200SpMotorstarterInterfaceAllUnits[0].EMmotorstarter[5].et200SpMotorstarterOutputs[0..1].reserve7 := FALSE;
   Et200SpMotorstarterInterfaceAllUnits[0].EMmotorstarter[6].et200SpMotorstarterOutputs[0..1].reserve7 := FALSE;
   Et200SpMotorstarterInterfaceAllUnits[0].EMmotorstarter[7].et200SpMotorstarterOutputs[0..1].reserve7 := FALSE;
   Et200SpMotorstarterInterfaceAllUnits[0].EMmotorstarter[0].et200SpMotorstarterOutputs[0..1].reserve8 := FALSE;
   Et200SpMotorstarterInterfaceAllUnits[0].EMmotorstarter[1].et200SpMotorstarterOutputs[0..1].reserve8 := FALSE;
   Et200SpMotorstarterInterfaceAllUnits[0].EMmotorstarter[2].et200SpMotorstarterOutputs[0..1].reserve8 := FALSE;
   Et200SpMotorstarterInterfaceAllUnits[0].EMmotorstarter[3].et200SpMotorstarterOutputs[0..1].reserve8 := FALSE;
   Et200SpMotorstarterInterfaceAllUnits[0].EMmotorstarter[4].et200SpMotorstarterOutputs[0..1].reserve8 := FALSE;
   Et200SpMotorstarterInterfaceAllUnits[0].EMmotorstarter[5].et200SpMotorstarterOutputs[0..1].reserve8 := FALSE;
   Et200SpMotorstarterInterfaceAllUnits[0].EMmotorstarter[6].et200SpMotorstarterOutputs[0..1].reserve8 := FALSE;
   Et200SpMotorstarterInterfaceAllUnits[0].EMmotorstarter[7].et200SpMotorstarterOutputs[0..1].reserve8 := FALSE;
   Et200SpMotorstarterInterfaceAllUnits[0].EMmotorstarter[0].et200SpMotorstarterOutputs[0..1].reserve9 := FALSE;
   Et200SpMotorstarterInterfaceAllUnits[0].EMmotorstarter[1].et200SpMotorstarterOutputs[0..1].reserve9 := FALSE;
   Et200SpMotorstarterInterfaceAllUnits[0].EMmotorstarter[2].et200SpMotorstarterOutputs[0..1].reserve9 := FALSE;
   Et200SpMotorstarterInterfaceAllUnits[0].EMmotorstarter[3].et200SpMotorstarterOutputs[0..1].reserve9 := FALSE;
   Et200SpMotorstarterInterfaceAllUnits[0].EMmotorstarter[4].et200SpMotorstarterOutputs[0..1].reserve9 := FALSE;
   Et200SpMotorstarterInterfaceAllUnits[0].EMmotorstarter[5].et200SpMotorstarterOutputs[0..1].reserve9 := FALSE;
   Et200SpMotorstarterInterfaceAllUnits[0].EMmotorstarter[6].et200SpMotorstarterOutputs[0..1].reserve9 := FALSE;
   Et200SpMotorstarterInterfaceAllUnits[0].EMmotorstarter[7].et200SpMotorstarterOutputs[0..1].reserve9 := FALSE;
   Et200SpMotorstarterInterfaceAllUnits[0].EMmotorstarter[0].et200SpMotorstarterOutputs[0..1].reserve10 := FALSE;
   Et200SpMotorstarterInterfaceAllUnits[0].EMmotorstarter[1].et200SpMotorstarterOutputs[0..1].reserve10 := FALSE;
   Et200SpMotorstarterInterfaceAllUnits[0].EMmotorstarter[2].et200SpMotorstarterOutputs[0..1].reserve10 := FALSE;
   Et200SpMotorstarterInterfaceAllUnits[0].EMmotorstarter[3].et200SpMotorstarterOutputs[0..1].reserve10 := FALSE;
   Et200SpMotorstarterInterfaceAllUnits[0].EMmotorstarter[4].et200SpMotorstarterOutputs[0..1].reserve10 := FALSE;
   Et200SpMotorstarterInterfaceAllUnits[0].EMmotorstarter[5].et200SpMotorstarterOutputs[0..1].reserve10 := FALSE;
   Et200SpMotorstarterInterfaceAllUnits[0].EMmotorstarter[6].et200SpMotorstarterOutputs[0..1].reserve10 := FALSE;
   Et200SpMotorstarterInterfaceAllUnits[0].EMmotorstarter[7].et200SpMotorstarterOutputs[0..1].reserve10 := FALSE;
   Et200SpMotorstarterInterfaceAllUnits[0].EMmotorstarter[0].et200SpMotorstarterOutputs[0..1].disableQuickStop := FALSE;
   Et200SpMotorstarterInterfaceAllUnits[0].EMmotorstarter[1].et200SpMotorstarterOutputs[0..1].disableQuickStop := FALSE;
   Et200SpMotorstarterInterfaceAllUnits[0].EMmotorstarter[2].et200SpMotorstarterOutputs[0..1].disableQuickStop := FALSE;
   Et200SpMotorstarterInterfaceAllUnits[0].EMmotorstarter[3].et200SpMotorstarterOutputs[0..1].disableQuickStop := FALSE;
   Et200SpMotorstarterInterfaceAllUnits[0].EMmotorstarter[4].et200SpMotorstarterOutputs[0..1].disableQuickStop := FALSE;
   Et200SpMotorstarterInterfaceAllUnits[0].EMmotorstarter[5].et200SpMotorstarterOutputs[0..1].disableQuickStop := FALSE;
   Et200SpMotorstarterInterfaceAllUnits[0].EMmotorstarter[6].et200SpMotorstarterOutputs[0..1].disableQuickStop := FALSE;
   Et200SpMotorstarterInterfaceAllUnits[0].EMmotorstarter[7].et200SpMotorstarterOutputs[0..1].disableQuickStop := FALSE;
END_DATA_BLOCK
